INTERFACE I_ControlBox

METHOD Lamps 
VAR_INPUT
	bEnable : BOOL;
END_VAR
END_METHOD

METHOD ModeSelector 
VAR_INPUT
END_VAR
VAR_OUTPUT
	eMode : E_Mode;
END_VAR
END_METHOD

END_INTERFACE

(* stored: Version 1.1.0.1, ProductVersion 3.1.4024.10
   Itf I_ControlBox: Id {5c741758-32b4-4a5c-b560-a63e85cb966e}
   Method Lamps: Id {705895e4-a55f-468b-bff0-8eb1edb6385c}
   Method ModeSelector: Id {602723b8-14f8-4c4d-9a3a-6c04bf063cdf} *)
